Staubli VAL3: readDB.pgx

public program readDB(num x_nDBnumber, num& x_nDB[])
  local num l_nLength
begin

  call getDBsize(x_nDBnumber, l_nLength)

  if nLastError==nNoErrors
    resize(x_nDB, 1, l_nLength)
    call readArea(nAreaDB, x_nDBnumber, 0, l_nLength, x_nDB)
  endIf

end
